(* PLC project Interface Example.project, CODESYS CODESYS V3.5 SP20 Patch 1 *)
(* stored: creationDateTime 2025-05-26T20:47:46.5927715, modificationDateTime 2025-05-26T20:46:17.1216239 *)

INTERFACE IMotor
METHOD Start : BOOL
END_METHOD
METHOD Stop : BOOL
END_METHOD
PROPERTY IsRunning : BOOL
END_PROPERTY
END_INTERFACE

PROGRAM Main
  VAR_INPUT
    Motor : IMotor;
  END_VAR

                    
// Call a method
Motor.Start();

// Get a property
IF Motor.IsRunning THEN (**) END_IF
                  
END_PROGRAM

FUNCTION_BLOCK Motor IMPLEMENTS IMotor

                    
// Motor control logic here
                  

METHOD Start : BOOL
                          
                        
END_METHOD

METHOD Stop : BOOL
                          
                        
END_METHOD

PROPERTY IsRunning : BOOL
GET
                            
                          
END_GET
SET
                            
                          
END_SET
END_PROPERTY
END_FUNCTION_BLOCK

CONFIGURATION Device
  RESOURCE Application ON PLC
    TASK MainTask(INTERVAL := T#20ms, PRIORITY := 1);
    PROGRAM Main WITH MainTask : Main;
  END_RESOURCE
END_CONFIGURATION
